{attribute addProperty BoxType "KL2284"}
{attribute addProperty Id "Channel_1Channel_9E062D1C00Channel_2Channel_9E062D1C00Channel_3Channel_9E062D1C00Channel_4Channel_9E062D1C00"}
{attribute addProperty CRC "4128136836"}
{attribute addProperty SizeInBites "0"}
{attribute addProperty SizeInBytes "0"}
TYPE KL2284_F60E5E84 :
STRUCT
	{attribute addProperty Name "Channel_1"}
	Channel_1 : Channel_9E062D1C;
	{attribute addProperty Name "Channel_2"}
	Channel_2 : Channel_9E062D1C;
	{attribute addProperty Name "Channel_3"}
	Channel_3 : Channel_9E062D1C;
	{attribute addProperty Name "Channel_4"}
	Channel_4 : Channel_9E062D1C;
END_STRUCT
END_TYPE

(* stored: Version 1.2.0.0, ProductVersion 3.1.4024.9
   DUT KL2284_F60E5E84: Id {278fc8fd-7b30-4652-a0bc-aa33037218c3} *)
